// TIA Portal V15.1 export
// export: Created 2026-01-15T16:29:47.0494675Z, ExportSetting WithDefaults, WithReadOnly, DisplayName Totally Integrated Automation Portal, DisplayVersion V15.1 Update 8, DisplayName TIA Portal Openness, DisplayVersion V15.1 Update 8, DisplayName STEP 7 Professional, DisplayVersion V15.1 Update 8, DisplayName WinCC Advanced, DisplayVersion V15.1 Update 8
FUNCTION "FCCA_CCD_AP1" : Void   // FC16, LAD
{ S7_Optimized_Access := 'TRUE' }
VERSION : 0.1
// stored: AutoNumber true, CodeModifiedDate 2026-01-15T16:25:54.3671983Z, CompileDate 2026-01-15T16:25:54.4076417Z, CreationDate 2026-01-15T16:24:02.4619467Z, HandleErrorsWithinBlock false, InterfaceModifiedDate 2024-08-08T03:24:33.8704482Z, IsConsistent true, IsIECCheckEnabled false, IsKnowHowProtected false, IsWriteProtected false, LibraryConformanceStatus Error: The block contains calls of single instances. Warning: The object contains access to global data blocks. Warning: The block contains direct access to inputs, outputs, bit memories, indirect access to the registry or indirect access to external memory areas that are unknown at the time of compilation., ModifiedDate 2026-01-15T16:25:54.3671983Z, ParameterModified 2024-08-08T03:24:33.8704482Z, PLCSimAdvancedSupport false, SetENOAutomatically False, StructureModified 2024-08-08T03:24:33.8704482Z, UDAEnableTagReadback false
BEGIN

REGION Network 1: Trạng thái cân Nước 1 hoặc AP1
   // Đầu tiên nó sẽ đợi một khoảng thời gian gọi là Thời gian trễ cân, sau đó nó mới đủ điều kiện để cân
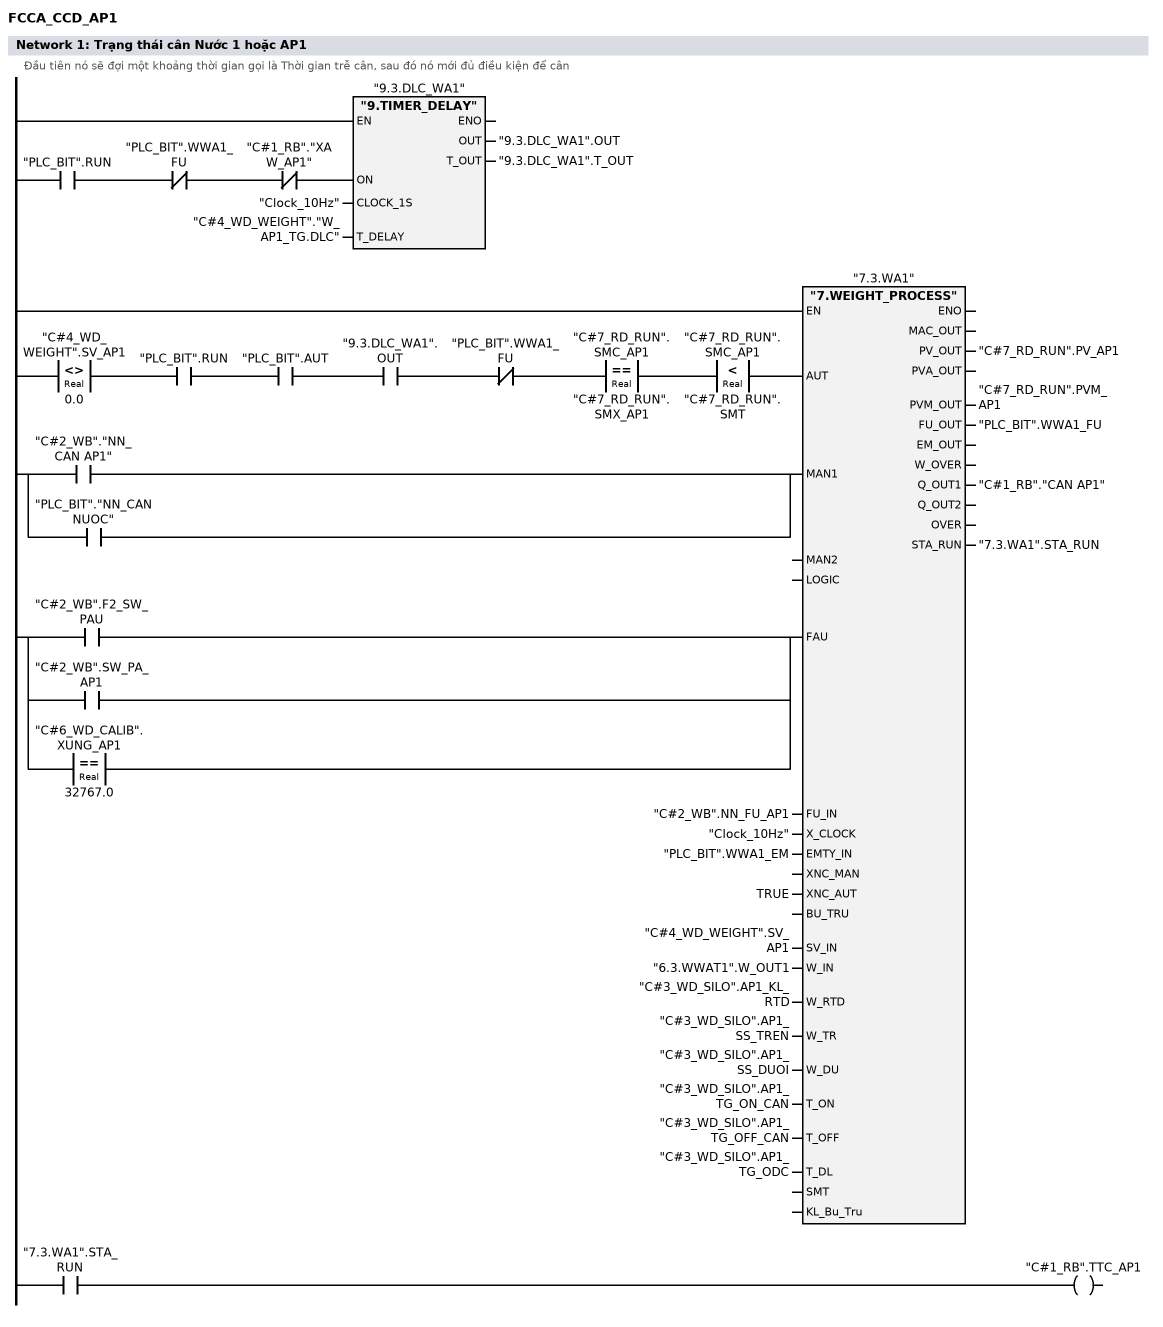
   RUNG wire#powerrail
      "9.3.DLC_WA1"(ON := wire#w1, CLOCK_1S := "Clock_10Hz", T_DELAY := "C#4_WD_WEIGHT"."W_AP1_TG.DLC", OUT => "9.3.DLC_WA1".OUT, T_OUT => "9.3.DLC_WA1".T_OUT)
   END_RUNG
   RUNG wire#powerrail
      Contact( "PLC_BIT".RUN )
      I_Contact( "PLC_BIT".WWA1_FU )
      I_Contact( "C#1_RB"."XA W_AP1" )
   END_RUNG wire#w1
   RUNG wire#powerrail
      "7.3.WA1"(AUT := wire#w2, MAN1 := wire#w3, FAU := wire#w4, MAN2 :=, LOGIC :=, FU_IN := "C#2_WB".NN_FU_AP1, X_CLOCK := "Clock_10Hz", EMTY_IN := "PLC_BIT".WWA1_EM, XNC_MAN :=, XNC_AUT := TRUE, BU_TRU :=, SV_IN := "C#4_WD_WEIGHT".SV_AP1, W_IN := "6.3.WWAT1".W_OUT1, W_RTD := "C#3_WD_SILO".AP1_KL_RTD, W_TR := "C#3_WD_SILO".AP1_SS_TREN, W_DU := "C#3_WD_SILO".AP1_SS_DUOI, T_ON := "C#3_WD_SILO".AP1_TG_ON_CAN, T_OFF := "C#3_WD_SILO".AP1_TG_OFF_CAN, T_DL := "C#3_WD_SILO".AP1_TG_ODC, SMT :=, KL_Bu_Tru :=, MAC_OUT =>, PV_OUT => "C#7_RD_RUN".PV_AP1, PVA_OUT =>, PVM_OUT => "C#7_RD_RUN".PVM_AP1, FU_OUT => "PLC_BIT".WWA1_FU, EM_OUT =>, W_OVER =>, Q_OUT1 => "C#1_RB"."CAN AP1", Q_OUT2 =>, OVER =>, STA_RUN => "7.3.WA1".STA_RUN)
   END_RUNG
   RUNG wire#powerrail
      { S7_Templates := "SrcType := Real" } NE_Contact(in1 := "C#4_WD_WEIGHT".SV_AP1, in2 := 0.0)
      Contact( "PLC_BIT".RUN )
      Contact( "PLC_BIT".AUT )
      Contact( "9.3.DLC_WA1".OUT )
      I_Contact( "PLC_BIT".WWA1_FU )
      { S7_Templates := "SrcType := Real" } EQ_Contact(in1 := "C#7_RD_RUN".SMC_AP1, in2 := "C#7_RD_RUN".SMX_AP1)
      { S7_Templates := "SrcType := Real" } LT_Contact(in1 := "C#7_RD_RUN".SMC_AP1, in2 := "C#7_RD_RUN".SMT)
   END_RUNG wire#w2
   RUNG wire#powerrail
      Contact( "C#2_WB"."NN_CAN AP1" )
   END_RUNG wire#w3
   RUNG wire#powerrail
      Contact( "PLC_BIT"."NN_CAN NUOC" )
   END_RUNG wire#w3
   RUNG wire#powerrail
      Contact( "C#2_WB".F2_SW_PAU )
   END_RUNG wire#w4
   RUNG wire#powerrail
      Contact( "C#2_WB".SW_PA_AP1 )
   END_RUNG wire#w4
   RUNG wire#powerrail
      { S7_Templates := "SrcType := Real" } EQ_Contact(in1 := "C#6_WD_CALIB".XUNG_AP1, in2 := 32767.0)
   END_RUNG wire#w4
   RUNG wire#powerrail
      Contact( "7.3.WA1".STA_RUN )
      Coil( "C#1_RB".TTC_AP1 )
   END_RUNG
   // the same network as SCL:
   "9.3.DLC_WA1"(ON := "PLC_BIT".RUN AND NOT "PLC_BIT".WWA1_FU AND NOT "C#1_RB"."XA W_AP1",   // "9.TIMER_DELAY"
                 CLOCK_1S := "Clock_10Hz",
                 T_DELAY := "C#4_WD_WEIGHT"."W_AP1_TG.DLC",
                 OUT => "9.3.DLC_WA1".OUT,
                 T_OUT => "9.3.DLC_WA1".T_OUT);
   "7.3.WA1"(AUT := ("C#4_WD_WEIGHT".SV_AP1 <> 0.0) AND "PLC_BIT".RUN AND "PLC_BIT".AUT AND "9.3.DLC_WA1".OUT AND NOT "PLC_BIT".WWA1_FU AND ("C#7_RD_RUN".SMC_AP1 = "C#7_RD_RUN".SMX_AP1) AND ("C#7_RD_RUN".SMC_AP1 < "C#7_RD_RUN".SMT),   // "7.WEIGHT_PROCESS"
             MAN1 := "C#2_WB"."NN_CAN AP1" OR "PLC_BIT"."NN_CAN NUOC",
             FAU := "C#2_WB".F2_SW_PAU OR "C#2_WB".SW_PA_AP1 OR ("C#6_WD_CALIB".XUNG_AP1 = 32767.0),
             FU_IN := "C#2_WB".NN_FU_AP1,
             X_CLOCK := "Clock_10Hz",
             EMTY_IN := "PLC_BIT".WWA1_EM,
             XNC_AUT := TRUE,
             SV_IN := "C#4_WD_WEIGHT".SV_AP1,
             W_IN := "6.3.WWAT1".W_OUT1,
             W_RTD := "C#3_WD_SILO".AP1_KL_RTD,
             W_TR := "C#3_WD_SILO".AP1_SS_TREN,
             W_DU := "C#3_WD_SILO".AP1_SS_DUOI,
             T_ON := "C#3_WD_SILO".AP1_TG_ON_CAN,
             T_OFF := "C#3_WD_SILO".AP1_TG_OFF_CAN,
             T_DL := "C#3_WD_SILO".AP1_TG_ODC,
             PV_OUT => "C#7_RD_RUN".PV_AP1,
             PVM_OUT => "C#7_RD_RUN".PVM_AP1,
             FU_OUT => "PLC_BIT".WWA1_FU,
             Q_OUT1 => "C#1_RB"."CAN AP1",
             STA_RUN => "7.3.WA1".STA_RUN);
   "C#1_RB".TTC_AP1 := "7.3.WA1".STA_RUN;
END_REGION
END_FUNCTION
